(* IEC 61131-3 sources: linguist_for_iec_61131-3/samples/Structured Text, 3 files *)

(* ---- blinker.iec ---- *)
// blinker.iec — IEC 61131-3 Structured Text: function_block and program example

{attribute 'enable_dynamic_creation'}
type
    TrafficLight : (Red, Yellow, Green) := Red;
end_type

function_block Blinker
var_input
    Enable    : bool;
    Interval  : time := t#500ms;
end_var
var_output
    Output    : bool;
end_var
var
    _timer    : TON;
end_var

_timer(IN := Enable, PT := Interval);

if _timer.Q then
    Output := not Output;
    _timer(IN := false);
end_if;

end_function_block

program Main
var
    counter   : dint := 0;
    limit     : dint := 16#FF;
    flag      : bool := false;
    ratio     : lreal := 1.5e-3;
    addr      : byte at %QB0;
    msg       : string[80] := 'Hello, $'IEC 61131-3$'!';
    light     : TrafficLight;
    blinker   : Blinker;
end_var

blinker(Enable := true, Interval := t#250ms);

for counter := 0 to 9 do
    case light of
        Red    : light := Green;
        Green  : light := Yellow;
        Yellow : light := Red;
    end_case;
end_for;

while counter > 0 do
    counter := counter - 1;
end_while;

repeat
    flag := not flag;
    counter := counter + 1;
until counter >= 5
end_repeat;

if flag and (counter < limit) then
    addr := byte#16#A5;
elsif not flag then
    addr := 2#10101010;
else
    addr := 8#377;
end_if;

end_program

(* ---- pid_controller.iecst ---- *)
// pid_controller.iecst — IEC 61131-3 Structured Text: PID controller example

type
    PidParams : struct
        Kp       : lreal;
        Ki       : lreal;
        Kd       : lreal;
        OutMin   : lreal := -100.0;
        OutMax   : lreal :=  100.0;
    end_struct;
end_type

function_block PidController
var_input
    Enable      : bool;
    Setpoint    : lreal;
    ProcessVar  : lreal;
    Params      : PidParams;
    CycleTime   : time := t#10ms;
end_var
var_output
    Output      : lreal;
    Error       : lreal;
end_var
var
    _integral   : lreal;
    _prevError  : lreal;
    _dt         : lreal;
end_var

if not Enable then
    Output    := 0.0;
    _integral := 0.0;
    _prevError := 0.0;
    return;
end_if;

_dt    := lreal#TIME_TO_LREAL(CycleTime) / 1000.0;
Error  := Setpoint - ProcessVar;

_integral := _integral + Error * _dt;

// anti-windup: clamp integral contribution
if Params.Ki <> 0.0 then
    _integral := limit(_integral, Params.OutMin / Params.Ki, Params.OutMax / Params.Ki);
end_if;

Output := Params.Kp * Error
        + Params.Ki * _integral
        + Params.Kd * (Error - _prevError) / _dt;

Output     := limit(Output, Params.OutMin, Params.OutMax);
_prevError := Error;

end_function_block

program TemperatureControl
var
    pid      : PidController;
    params   : PidParams := (Kp := 2.5, Ki := 0.1, Kd := 0.05);
    setpoint : lreal := 75.0;
    measured : lreal at %IW0;
    heater   : lreal at %QW0;
end_var

pid(
    Enable     := true,
    Setpoint   := setpoint,
    ProcessVar := measured,
    Params     := params,
    CycleTime  := t#10ms
);

heater := pid.Output;

end_program

(* ---- tank_level.st ---- *)
(* tank_level.st - two-point level control with fill/drain valves and alarm text *)

type
    TankState : (Idle, Filling, Draining, Fault) := Idle;
end_type

function_block TankLevel
var_input
    Level      : real;          (* measured level in percent *)
    LowLimit   : real := 20.0;
    HighLimit  : real := 80.0;
    Reset      : bool;
end_var
var_output
    FillValve  : bool;
    DrainValve : bool;
    Alarm      : bool;
    Message    : string(80);
end_var
var
    State      : TankState;
    FaultTimer : TON;
end_var

FaultTimer(IN := (State = Filling) and (Level < LowLimit), PT := t#30s);

case State of
    Idle:
        if Level < LowLimit then
            State := Filling;
        elsif Level > HighLimit then
            State := Draining;
        end_if;
    Filling:
        if Level >= HighLimit then
            State := Idle;
        elsif FaultTimer.Q then
            State := Fault;
        end_if;
    Draining:
        if Level <= LowLimit then
            State := Idle;
        end_if;
    Fault:
        if Reset then
            State := Idle;
        end_if;
end_case;

FillValve  := State = Filling;
DrainValve := State = Draining;
Alarm      := State = Fault;

if Alarm then
    Message := 'Tank fill timeout$R$L';
else
    Message := '';
end_if;
end_function_block
